# EPICS substitutions: elioApp/Db/EL3068.substitutions
file EL3068.template { pattern
{ CHAN	}
{ 1	}
{ 2	}
{ 3	}
{ 4	}
{ 5	}
{ 6	}
{ 7	}
{ 8	}
}
